Staubli VAL3: clkEndProgram.pgx

program clkEndProgram()
begin
  bEndProgram = true
  bDoAirex    = false
  bDoModules  = false
  bGlueGlass  = false
end
